// TIA Portal V18 export
TYPE "AM CTRL"
// stored: IsFailsafeCompliant false
   STRUCT
      "AUTO/MAN" : Bool := TRUE;
      "MAN START" : Bool;
      "MAN STOP" : Bool;
   END_STRUCT;
END_TYPE
